# B&R Automation Studio project robot_control
Automation Studio 4.8.2.72

## Configuration Config1

CPU X20CP1382, AutomationRuntime B4.82, Build 4.1.2, Vc V4.72.1

### Hardware
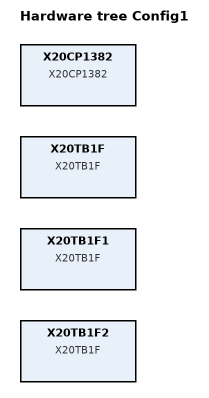
```
X20CP1382 : X20CP1382 v1.10.0.0  [X1 -> X1.SL; X2 -> X2.SL; X3 -> X3.SL]
  Module X1 (Type=X1, Virtual=true, Version=1.10.0.0)
    Connection (Connector=SS1, TargetModule=X20TB1F, TargetConnector=SS)
    Connection (Connector=SL, TargetModule=X20CP1382, TargetConnector=X1)
  Module X2 (Type=X2, Virtual=true, Version=1.10.0.0)
    Connection (Connector=SS1, TargetModule=X20TB1F1, TargetConnector=SS)
    Connection (Connector=SL, TargetModule=X20CP1382, TargetConnector=X2)
  Module X3 (Type=X3, Virtual=true, Version=1.10.0.0)
    Connection (Connector=SS1, TargetModule=X20TB1F2, TargetConnector=SS)
    Connection (Connector=SL, TargetModule=X20CP1382, TargetConnector=X3)
  Connector IF2:
    ActivateDevice = 1
    Mode = Manual
    InternetAddress = 10.0.0.50
    SubnetMask = 255.255.255.0
    ActivateSnmp = 2
  Connector IF7:
    Timeout = 1
  ConfigurationID = robot_control_Config1
  SystemTick = 1000
  Cyclic1Duration = 1000
X20TB1F : X20TB1F v1.0.0.0
X20TB1F1 : X20TB1F v1.0.0.0
X20TB1F2 : X20TB1F v1.0.0.0
```

### IoMap.iom - X20CP1382/IoMap.iom
```iecst
VAR_CONFIG
	::Program:this.M1.direction AT %QX."X3".DigitalOutput04;
	::Program:this.M1.freq AT %QX."X3".DigitalOutput09;
	::Program:this.M2.direction AT %QX."X3".DigitalOutput05;
	::Program:this.M3.direction AT %QX."X3".DigitalOutput06;
	::Program:this.M2.freq AT %QX."X3".DigitalOutput10;
	::Program:this.M3.freq AT %QX."X3".DigitalOutput11;
	::Program:this.btn1.pressed AT %IX."X1".DigitalInput03;
	::Program:this.btn2.pressed AT %IX."X1".DigitalInput02;
	::Program:this.btn4.pressed AT %IX."X1".DigitalInput04;
	::Program:this.btn3.pressed AT %IX."X1".DigitalInput01;
	::Program:this.pencilSharp AT %QX."X3".DigitalOutput08;
END_VAR
```

## Logical view

Binary libraries used (declarations not repeated): operator, runtime, astime, AsIecCon, AsOpcUac, AsOpcUas, AsTCP, AsBrStr

### Global.var - Global variables
```iecst
VAR
	SPEED : TIME;
	gNettime : DINT;
	pSharp : BOOL;
	draw_old : DINT;
	draw : DINT := 0;
	y_coord : DINT := 0;
	x_coord : DINT := 0;
	goTo : STRING[80];
END_VAR
```


### Program Logical/Program (IEC)

#### Types.typ
```iecst
TYPE
	m_typ : 	STRUCT
		endSwitch : BOOL;
		freq1 : BOOL;
		freq : BOOL;
		backward : BOOL;
		forward : BOOL;
		direction : BOOL;
		counter : DINT;
		goTo : BOOL;
		goToCounter : DINT;
		speedCase : USINT;
	END_STRUCT;
	this_typ : 	STRUCT
		M2 : m_typ;
		M3 : m_typ;
		M1 : m_typ;
		btn2 : btn_typ;
		isReady : BOOL;
		btn4 : btn_typ;
		btn3 : btn_typ;
		btn1 : btn_typ;
		startCase : USINT;
		start : BOOL;
		startPSCase : USINT;
		startPS : BOOL;
		pencilSharp : BOOL;
	END_STRUCT;
	btn_typ : 	STRUCT
		pressed : BOOL;
	END_STRUCT;
END_TYPE
```

#### Variables.var
```iecst
VAR
	dull_counter : DINT;
	sharp_counter2 : DINT;
	sharp_counter : DINT;
	case_draw : USINT;
	this : this_typ;
END_VAR
```

#### Main.st
```iecst
PROGRAM _INIT
	draw := 5;
	this.start := TRUE;
	this.topSpeed 		:= T#0ms; 	// This parameter will slow the topspeed of all axis.
	this.acceleration	:= 1;		// This parameter will smoothen the acceleration of all axis.

END_PROGRAM

PROGRAM _CYCLIC
	(**********************************************************************************************)
	(************************************** Startup sequence **************************************)
	(**********************************************************************************************)
	IF this.start AND gNettime <> 0 THEN
		CASE this.startCase OF
			0: // First find M3 and M2 home switch
				this.M3.backward 	:= TRUE;
				this.M2.backward 	:= TRUE;

				IF this.btn3.pressed THEN
					this.M1.backward:= TRUE;
					this.startCase 	:= 10;
				END_IF;

			10: // Waiting for M1 and M2 to be homed
				IF this.btn1.pressed THEN
					this.M1.counter	:= 0;
				END_IF;

				IF this.btn2.pressed THEN
					this.M2.counter := 0;
				END_IF;

				IF this.btn1.pressed AND this.btn2.pressed THEN
					this.startCase := 15;
				END_IF;

			15:// going to origo (0,0)
				IF this.M1.counter < 4000 THEN
					this.M1.forward := TRUE;
				ELSE
					this.M1.forward := FALSE;
				END_IF;

				IF this.M2.counter < 150 THEN
					this.M2.forward := TRUE;
				ELSE
					this.M2.forward := FALSE;
				END_IF;

				IF this.M1.counter >= 4000 AND this.M2.counter >= 150 THEN
					this.startCase := 20;
				END_IF;

			20: // make sure the pencil have reached origo with M3
				IF this.btn4.pressed THEN
					this.startCase := 25;
				ELSE
					this.M3.forward := TRUE;
				END_IF;

			25: // Set all counter values to 0
				this.M1.counter := 0;
				this.M2.counter := 0;
				this.M3.counter := 0;
				this.startCase := 30;

			30: // Lift the pencil from the paper again
				IF this.M3.counter > -500 THEN
					this.M3.backward := TRUE;
				ELSE
					this.M3.backward := FALSE;
					this.startCase := 35;
				END_IF;

			35: // Ready to start drawing
				this.start 		:= FALSE;
				this.startCase 	:= FALSE;
				this.isReady 	:= TRUE;

		END_CASE;
	END_IF

	(**********************************************************************************************)
	(*********************************** Coordinate translation ***********************************)
	(**********************************************************************************************)
	// Read and translate the coordinates from java server
	IF NOT pSharp THEN
		CASE case_draw OF
			0: // start the case
				IF coord[LENGT_OF_COORD].x <> -1 AND coord[LENGT_OF_COORD].y <> -1 AND coord[LENGT_OF_COORD].z <> -1 THEN
					this.coord.x := coord[LENGT_OF_COORD].x;
					this.coord.y := coord[LENGT_OF_COORD].y;
					this.coord.z := coord[LENGT_OF_COORD].z;
					coord[LENGT_OF_COORD].x := -1;
					coord[LENGT_OF_COORD].y := -1;
					coord[LENGT_OF_COORD].z := -1;
					case_draw := 5;
				END_IF

			5: // which height should we goto?
				IF this.coord.z = 0 THEN // Black
					this.M3.goToCounter := 110;
					this.M3.goTo 		:= TRUE;
				ELSIF this.coord.z = 1 THEN
					this.M3.goToCounter := 75;
					this.M3.goTo 		:= TRUE;
				ELSIF this.coord.z = 2 THEN
					this.M3.goToCounter := 30;
					this.M3.goTo 		:= TRUE;
				ELSIF this.coord.z = 3 THEN
					this.M3.goToCounter := -65;
					this.M3.goTo 		:= TRUE;
				ELSIF this.coord.z = 4 THEN
					this.M3.goToCounter := -71;
					this.M3.goTo 		:= TRUE;
				ELSIF this.coord.z = 5 THEN // White
					this.M3.goToCounter := -110;
					this.M3.goTo 		:= TRUE;
				END_IF

				IF this.M3.counter = this.M3.goToCounter THEN
					case_draw := 10;
				END_IF

			10: // Goto all the coordinates, and then go back to state 0 to calculate next coordinate
				this.M1.goToCounter := this.coord.x * 40;
				this.M2.goToCounter := this.coord.y * 40;
				this.M1.goTo := TRUE;
				this.M2.goTo := TRUE;
				IF this.M3.counter <> this.M3.goToCounter THEN
					this.M3.goTo := TRUE;
				END_IF

				IF (this.M1.goToCounter = this.M1.counter AND this.M2.goToCounter = this.M2.counter AND this.M3.goToCounter = this.M3.counter) THEN
					case_draw := 0;
				END_IF

		END_CASE;
	END_IF;

	(**********************************************************************************************)
	(*********************************** Pencil sharpener logic ***********************************)
	(**********************************************************************************************)
	// Controls the acceleration when pencil sharpening
	IF EDGEPOS(pSharp) AND this.acceleration < 2 THEN
		this.acceleration 			:= this.acceleration + 2;
		this.accelerationChangePS 	:= TRUE;
	ELSIF EDGENEG(pSharp) AND this.accelerationChangePS THEN
		this.acceleration			:= this.acceleration - 2;
		this.accelerationChangePS	:= FALSE;
	END_IF

	// Calculate when to sharp the pencil
	// No wear on the pencil when draw value is 5
	// Approx. 175000 ms if the pencil draw value is 4
	// Approx. 164000 ms if the pencil draw value is 3
	// Approx. 150000 ms if the pencil draw value is 2
	// Approx. 130000 ms if the pencil draw value is 1
	// Approx. 100000 ms if the pencil draw value is 0

	IF draw = 4 THEN
		dull_counter := dull_counter + 1;
	ELSIF draw = 3 THEN
		dull_counter := dull_counter + 1.06;
	ELSIF draw = 2 THEN
		dull_counter := dull_counter + 1.16;
	ELSIF draw = 1 THEN
		dull_counter := dull_counter + 1.35;
	ELSIF draw = 0 THEN
		dull_counter := dull_counter + 1.75;
	END_IF

	IF (dull_counter > 175000) THEN
		pSharp := TRUE;
		dull_counter := 0;
		this.startPS := TRUE;
	END_IF;

	IF this.startPS THEN // When the dull counter runs out, pencil sharpener case starts
		CASE this.startPSCase OF
			0: // Store goTo values
				this.M1.goToCounter := this.M1.counter;
				this.M3.goToCounter := this.M3.counter;
				this.m3TempPS		:= this.M3.counter;
				this.startPSCase := 5;

			5: // lift the pencil from the drawing plane, and go to an height that fits the pencil sharpener
				this.M3.backward := TRUE;

				IF this.M3.counter < -200 AND this.M1.counter > -2500 THEN
					this.M1.backward := TRUE;
				ELSE
					this.M1.backward := FALSE;
				END_IF

				IF this.M3.counter = -3200 THEN
					this.M3.backward := FALSE;
					this.startPSCase := 10;
				END_IF

			10: // Start moving towards the pencil sharpener, and wait for switch above pencil sharpener to be activated
				this.M1.backward := TRUE;
				IF this.btn1.pressed THEN
					this.M1.backward := FALSE;
					this.startPSCase := 15;
				END_IF

			15: // start pencil sharpener, and go into the pencil sharpener
				this.pencilSharp := TRUE;
				this.M3.goToCounter := 110;
				this.M3.goTo := TRUE;

				IF EDGEPOS(this.btn4.pressed)THEN
					this.M3.counter	:= 0;
				END_IF

				IF this.btn4.pressed THEN
					sharp_counter := sharp_counter +1;
				END_IF

				IF sharp_counter > 500 THEN // go deeper
					sharp_counter := 0;
					this.startPSCase := 16;
				END_IF;

			16: // start going deeper
				this.M3.goToCounter := 130;
				this.M3.goTo := TRUE;
				sharp_counter := sharp_counter +1;

				IF sharp_counter > 500 THEN // go deeper
					sharp_counter := 0;
					this.startPSCase := 17;
				END_IF;

			17: // start going deeper
				this.M3.goToCounter := 145;
				this.M3.goTo := TRUE;
				sharp_counter := sharp_counter +1;

				IF sharp_counter > 3000 THEN // retreat
					sharp_counter := 0;
					this.startPSCase := 20;
				END_IF;

			20: // move out of the pencil sharpener
				this.M3.backward := TRUE;

				IF this.M3.counter = -1950 THEN
					this.M3.backward := FALSE;
					this.startPSCase := 25;
					this.pencilSharp := FALSE;
				END_IF

			25: // move back to position
				this.M1.goTo := TRUE;

				IF this.M1.counter > - 2800 THEN
					this.M3.goToCounter := 900;
					this.M3.goTo 		:= TRUE;
					this.startPSCase 	:= 27;
				END_IF

			27: // Calibrate axis 3 on the drawining plane
				IF this.M1.goTo = FALSE AND this.M3.goTo = FALSE THEN
					this.M3.forward := TRUE;
				END_IF

				IF this.btn4.pressed THEN
					this.M3.counter 	:= 0;
					this.M3.forward		:= FALSE;
					this.startPSCase 	:= 30;
				END_IF

			30: // go to the correct heigt
				IF this.M1.goTo = FALSE THEN
					this.M3.goToCounter := this.m3TempPS;
					this.M3.goTo := TRUE;
					this.startPSCase := 35;
				END_IF

			35: // Continues from where it left
				this.startPS := FALSE;
				this.startPSCase := 0;
				pSharp := FALSE;

		END_CASE
	END_IF

	(**********************************************************************************************)
	(****************************************** Subcasses *****************************************)
	(**********************************************************************************************)
	M1_speedCase;
	M2_speedCase;
	M3_speedCase;

END_PROGRAM
```

### Program Logical/TCPServer (IEC)

#### Variables.var
```iecst
VAR
	elPreben : BOOL; (*The most overpowered bollean expression on Funen*)
	F_It_TON : TON;
	coord_counter : USINT;
	TcpClose2 : TcpClose;
	TcpClose1 : TcpClose;
	TcpSend1 : TcpSend;
	TcpReceive1 : TcpRecv;
	TcpServer1 : TcpServer;
	TcpOpen1 : TcpOpen;
	receiveData : STRING[80];
	sendData : STRING[80];
	tcpst : TCPSTATE;
END_VAR
```

#### Main.st
```iecst
PROGRAM _INIT
	tcpst := TCPSTATE_SOCKET_OPEN;
	coord_counter := 1;
	x_coord := 0;
	y_coord := 0;
	draw := 0;
	sendData := '';
	receiveData := '';
	goTo := '';
	END_PROGRAM

PROGRAM _CYCLIC
	CASE tcpst OF
		TCPSTATE_SOCKET_OPEN :
			TcpOpen1.enable := TRUE;
			TcpOpen1.port := 12345;
			TcpOpen1.options := tcpOPT_REUSEADDR;
			TcpOpen1();
			IF (TcpOpen1.status = ERR_OK) OR (TcpOpen1.status = 32600) THEN
				tcpst := TCPSTATE_SERVER_CREATE;
			END_IF

		TCPSTATE_SERVER_CREATE :
			IF goTo = sendData AND goTo = receiveData AND goTo <> '' THEN
				IF coord_counter = 1 THEN
					x_coord := brsatoi(ADR(goTo));
				ELSIF coord_counter = 2 THEN
					y_coord := brsatoi(ADR(goTo));
				ELSIF coord_counter = 3 THEN
					draw := brsatoi(ADR(goTo));
				END_IF
				sendData := receiveData := '';
				// goTo := '';
				coord_counter := coord_counter + 1;
				IF coord_counter >= 4 THEN
					coord_counter := 1;
					goTo := 'ready';
					elPreben := TRUE;
				END_IF

			END_IF;
			IF NOT pSharp THEN
				IF goTo = 'done' THEN
					sendData := goTo;
					// goTo := '';
					tcpst := TCPSTATE_SEND;
				END_IF;
			END_IF;
			TcpServer1.enable := TRUE;
			TcpServer1.ident := TcpOpen1.ident;
			TcpServer1();
			IF (TcpServer1.status = ERR_OK) OR (TcpServer1.status = 32600) THEN
				tcpst := TCPSTATE_RECEIVE;
			END_IF

		TCPSTATE_RECEIVE :
			IF goTo = 'done' THEN
				tcpst := TCPSTATE_SERVER_CREATE;
			ELSIF goTo = '' AND elPreben = TRUE THEN
				F_It_TON.PT 	:= T#5000ms;
				F_It_TON.IN 	:= TRUE;

				IF F_It_TON.Q THEN
					goTo 		:= 'done';
					elPreben 	:= FALSE;
					F_It_TON.IN := TRUE;
				END_IF
			END_IF

			TcpReceive1.enable := TRUE;
			TcpReceive1.ident := TcpServer1.identclnt;
			TcpReceive1.pData := ADR(receiveData);
			TcpReceive1.datamax := SIZEOF(receiveData);
			TcpReceive1();
			IF (TcpReceive1.status = ERR_OK) OR (TcpReceive1.status = 32600) THEN
				tcpst := TCPSTATE_SEND;
				sendData := receiveData;
			END_IF

		TCPSTATE_SEND :
			TcpSend1.enable := TRUE;
			TcpSend1.ident := TcpServer1.identclnt;
			TcpSend1.pData := ADR(sendData);
			TcpSend1.datalen := brsstrlen(ADR(sendData));     // We use brsstrlen() to get the length in UDINT datatype
			TcpSend1();
			IF (TcpSend1.status = ERR_OK) OR (TcpSend1.status = 32600) THEN
				tcpst := TCPSTATE_CLOSE;
			END_IF

		TCPSTATE_CLOSE :
			goTo := sendData;
			IF sendData = 'done' THEN
				sendData := '';
			END_IF;
			TcpClose1.enable := TRUE;
			TcpClose1.ident := TcpServer1.identclnt;
			TcpClose1();
			IF (TcpClose1.status = ERR_OK) OR (TcpClose1.status = 32600) THEN
				TcpServer1.enable := FALSE;
				TcpServer1();
				tcpst := TCPSTATE_SERVER_CREATE;
			END_IF

	END_CASE

	IF tcpst <> TCPSTATE_RECEIVE THEN
		F_It_TON.IN := FALSE;
	END_IF

	F_It_TON();

	END_PROGRAM

PROGRAM _EXIT
	TcpClose1.enable := TRUE;
	TcpClose1.ident := TcpServer1.identclnt;
	TcpClose1();

	TcpClose2.enable := TRUE;
	TcpClose2.ident := TcpOpen1.ident;
	TcpClose2();
	END_PROGRAM
```

Listed in the project but not available here: Logical/Global.typ, Logical/OpcUA
